//{attribute 'qualified_only'}
VAR_GLOBAL CONSTANT
// HAUD 2023 12 13
  Version             : STRING  := '3.2.1';


  MAX_MOVER           : UINT    := 7;
  MAX_GROUP           : UINT    := 1;
END_VAR

(* stored: Version 1.1.0.1, ProductVersion 3.1.4024.12
   GVL XTS_Parameter: Id {926495ad-a98c-489a-a36b-a136e7e2c25a}, ParameterList True *)
